FUNCTION_BLOCK FB_CollectCPUData
VAR
	bFirstCycle				: BOOL := TRUE;	// First cycle of Function Call
	bExecuteRead 			: BOOL;
	tPeriod 				: TIME := T#500MS ;

	fbReadIPCTemperature 	: FB_IPCDiag_ReadParameterPeriodic 	;
	
	fbReadIPCUsage		 	: FB_IPCDiag_ReadParameterPeriodic 	;
	tInterval				: TIME := T#0.5S ; // Read interval
	
	
	stCPUData				: ST_CPUData ;
	fbDiagRegister			: FB_IPCDiag_Register ;
	
	stTaskData				: ST_TaskData;
	fbTcSyslatency			: TC_SysLatencyEx;
	
	arBuffer					: ARRAY [0..100] OF DINT ; 
	
	
END_VAR

// Initiate IPC diagnostics register
fbDiagRegister(bExecute := bFirstCycle);

IF fbDiagRegister.bValid THEN 
	bFirstCycle 	:= FALSE;
	bExecuteRead 	:= TRUE; 
END_IF

// Read and process data
mReadTemperatureData(); 
mReadCPUUsageData();

PROPERTY PUBLIC GetCPUData : ST_CPUData
GET
GetCPUData := stCPUData;
END_GET
END_PROPERTY

PROPERTY PUBLIC GetTaskData : ST_TaskData
GET
GetTaskData := stTaskData;
END_GET
END_PROPERTY

METHOD PRIVATE mReadCPUUsageData : ST_CPUUsage
VAR
	nCPUUsage				: UINT ; // current cPU usage [%] 
	TaskIndex		: DINT ; // current task index
END_VAR
// read temperature diagnostic data
fbReadIPCUsage(
	bEnable:= TRUE, 
	eParameterKey:= E_IPCDiag_ParameterKey.CPU_Usage, 
	tPeriod:= T#1S, 
	fbRegister:= fbDiagRegister );

fbTcSyslatency(bExecute := fbReadIPCUsage.bValid);
	
// Process data
IF fbReadIPCUsage.bValid THEN 
	fbReadIPCUsage.GetParameter(pBuffer := ADR(nCPUUsage), nBufferSize := SIZEOF(nCPUUsage)) ;
	stCPUData.stUsageData.nCPUUsage		:= nCPUUsage;
	stCPUData.stUsageData.nMaxCPUUsage 	:= MAX(nCPUUsage, stCPUData.stUsageData.nMaxCPUUsage);
	stCPUData.stUsageData.nCPUOverload	:= nCPUUsage > stCPUData.stUsageData.nLimitCPUUsage;

	TaskIndex := GETCURTASKINDEXEX();
	stTaskData.CycleTime	:= _TaskInfo[TaskIndex].CycleTime / 10000.0; //convert 100ns to ms
	stTaskData.LastExecTime	:= _TaskInfo[TaskIndex].LastExecTime / 10000.0; //convert 100ns to ms
	stTaskData.SystemLatency:= fbTcSyslatency.nActual;
END_IF
END_METHOD

METHOD PRIVATE mReadTemperatureData : ST_CPUTemperature 
VAR
	nCPUTemperature : INT ;
END_VAR
// read temperature diagnostic data
fbReadIPCTemperature(
	bEnable:= bExecuteRead, 
	eParameterKey:= E_IPCDiag_ParameterKey.CPU_Temp, 
	tPeriod:= T#1S, 
	fbRegister:= fbDiagRegister );
	
// Process data
IF fbReadIPCTemperature.bValid THEN 
	fbReadIPCTemperature.GetParameter(pBuffer := ADR(nCPUTemperature), nBufferSize := SIZEOF(nCPUTemperature)) ;
	stCPUData.stTemperatureData.nCPUCurrentTemparature	:= nCPUTemperature;
	stCPUData.stTemperatureData.nCPUMaximumTemperature	:= MAX(nCPUTemperature, stCPUData.stTemperatureData.nCPUMaximumTemperature);
	stCPUData.stTemperatureData.bInThermalThrottling 	:= nCPUTemperature >= stCPUData.stTemperatureData.nCPUTemperatureLimit;
END_IF
END_METHOD

END_FUNCTION_BLOCK

(* stored: Version 1.1.0.1
   POU FB_CollectCPUData: Id {02ad8f84-0f29-478d-8375-c684dca63912}, SpecialFunc None
   Property GetCPUData: Id {ebd4c9e4-4031-4d7f-81d3-2831a538a4d9}
   Get Get: Id {42fd44c0-7ada-46c0-a401-554ca1225f19}
   Property GetTaskData: Id {0d2cfdd8-ce72-40cd-a6f9-fa8b32c08fc3}
   Get Get: Id {f61014ac-833d-4ba0-95ca-5a6e0c898bb3}
   Method mReadCPUUsageData: Id {ee4a5b7b-951b-4495-89cb-c730a9f11c6c}
   Method mReadTemperatureData: Id {ff03ba25-3a5e-481d-b49c-83d14f12199d} *)
